(* Schneider Machine Expert - Basic project Tank_1m_Ultrasonic_TM221CE16T, file version 3.0.0.0 *)
(* ProjectInformations: Name=Tank_1m_Ultrasonic_TM221CE16T *)

HARDWARE
  Cpu 0: TM221CE16T
  ModuleExtensionObject 0: TM3AI4/G
  EthernetConfiguration: NetworkName=M221, IpAllocationMode=FixedAddress, IpAddress=0.0.0.0, SubnetMask=0.0.0.0
  SerialLineConfiguration: Baud=Baud19200, Parity=ParityEven, DataBits=DataBits8, StopBits=StopBits1, PhysicalMedium=PhysicalMediumRs485, TransmissionMode=TransmissionModeModbusRtu, SlaveId=1, Addressing=SlaveAddressing
  MastTask: UsePeriodScanMode=false, PeriodScan=100
  FastTask: Period=255
  CpuBehavior: StartingMode=StartAsPreviousState, AutoSaveRamOnEeprom=true, WatchdogPeriod=250

SYMBOLS  (address, symbol, comment, settings)
  %M0       INLET_ENABLE
  %M1       OUTLET_ENABLE
  %M2       LEVEL_HIGH
  %M3       LEVEL_LOW
  %S12      SB_RUNMODE  "The controller is running"
  %MW0      TANK_RAW  "Raw analog value from ultrasonic sensor (0-10000)"
  %MW1      TANK_LEVEL_MM  "Calculated tank level in millimeters (0-1000)"
  %MW2      TANK_LITERS  "Tank volume in liters for HMI display (0-1000L)"
  %Q0.0     INLET_VALVE
  %Q0.1     OUTLET_VALVE
  %IW1.0    ULTRASONIC_LEVEL  [Type=Type_0_10V, Scope=Scope_Normal, Minimum=0, Maximum=10000]

POU Tank Level Control
  (* SectionNumber=0 *)

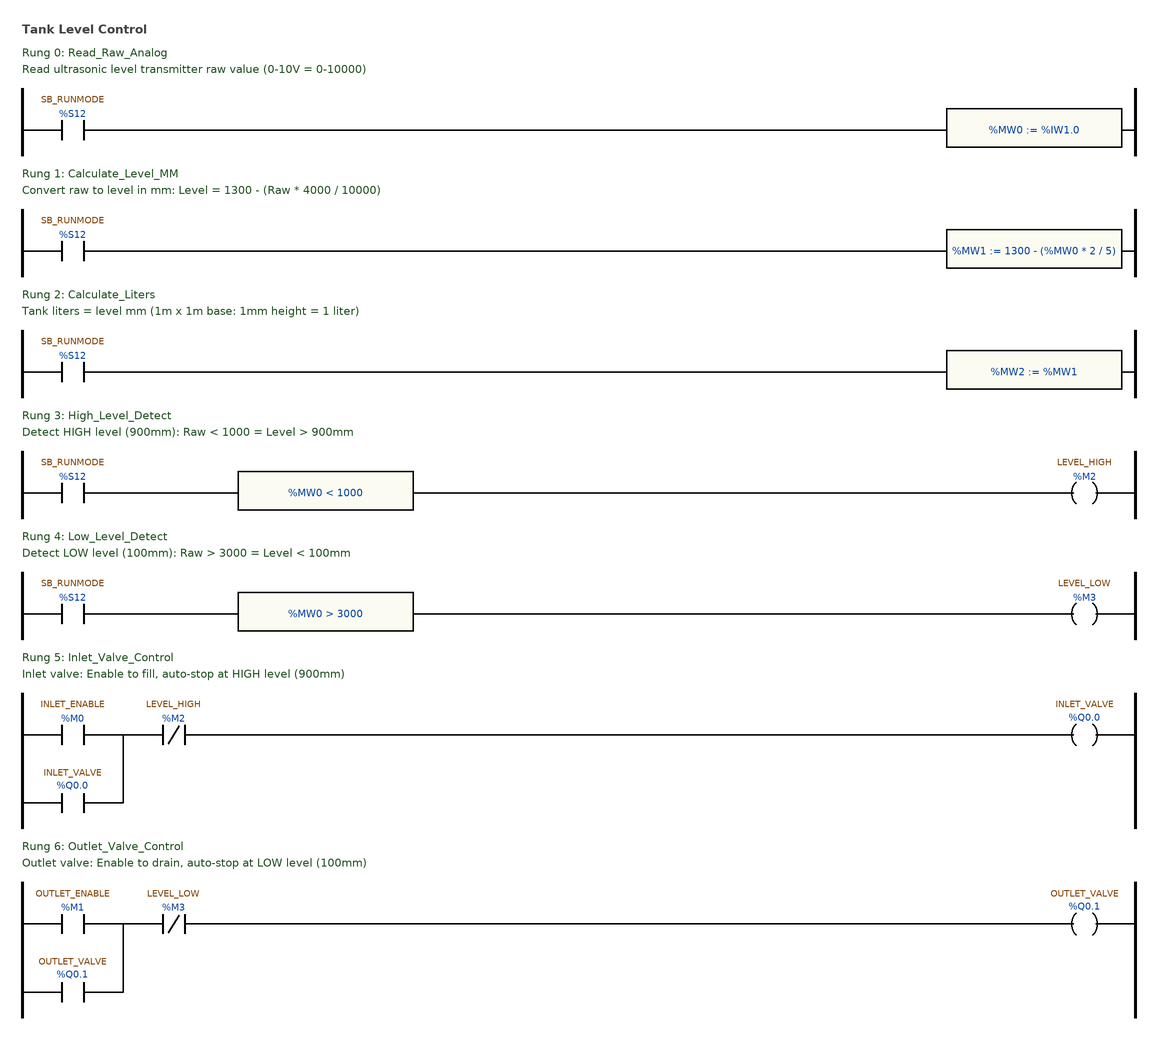

// Rung 0: Read_Raw_Analog
// Read ultrasonic level transmitter raw value (0-10V = 0-10000)
  LD %S12                 (* SB_RUNMODE *)
  [ %MW0 := %IW1.0 ]      (* TANK_RAW, ULTRASONIC_LEVEL *)
  // as ST:
  //   IF SB_RUNMODE THEN TANK_RAW := ULTRASONIC_LEVEL; END_IF;

// Rung 1: Calculate_Level_MM
// Convert raw to level in mm: Level = 1300 - (Raw * 4000 / 10000)
  LD %S12                 (* SB_RUNMODE *)
  [ %MW1 := 1300 - (%MW0 * 2 / 5) ](* TANK_LEVEL_MM, TANK_RAW *)
  // as ST:
  //   IF SB_RUNMODE THEN TANK_LEVEL_MM := 1300 - (TANK_RAW * 2 / 5); END_IF;

// Rung 2: Calculate_Liters
// Tank liters = level mm (1m x 1m base: 1mm height = 1 liter)
  LD %S12                 (* SB_RUNMODE *)
  [ %MW2 := %MW1 ]        (* TANK_LITERS, TANK_LEVEL_MM *)
  // as ST:
  //   IF SB_RUNMODE THEN TANK_LITERS := TANK_LEVEL_MM; END_IF;

// Rung 3: High_Level_Detect
// Detect HIGH level (900mm): Raw < 1000 = Level > 900mm
  LD %S12                 (* SB_RUNMODE *)
  AND [ %MW0 < 1000 ]     (* TANK_RAW *)
  ST %M2                  (* LEVEL_HIGH *)
  // as ST:
  //   LEVEL_HIGH := SB_RUNMODE AND TANK_RAW < 1000;

// Rung 4: Low_Level_Detect
// Detect LOW level (100mm): Raw > 3000 = Level < 100mm
  LD %S12                 (* SB_RUNMODE *)
  AND [ %MW0 > 3000 ]     (* TANK_RAW *)
  ST %M3                  (* LEVEL_LOW *)
  // as ST:
  //   LEVEL_LOW := SB_RUNMODE AND TANK_RAW > 3000;

// Rung 5: Inlet_Valve_Control
// Inlet valve: Enable to fill, auto-stop at HIGH level (900mm)
  LD %M0                  (* INLET_ENABLE *)
  OR %Q0.0                (* INLET_VALVE *)
  ANDN %M2                (* LEVEL_HIGH *)
  ST %Q0.0                (* INLET_VALVE *)
  // as ST:
  //   INLET_VALVE := (INLET_ENABLE OR INLET_VALVE) AND NOT LEVEL_HIGH;

// Rung 6: Outlet_Valve_Control
// Outlet valve: Enable to drain, auto-stop at LOW level (100mm)
  LD %M1                  (* OUTLET_ENABLE *)
  OR %Q0.1                (* OUTLET_VALVE *)
  ANDN %M3                (* LEVEL_LOW *)
  ST %Q0.1                (* OUTLET_VALVE *)
  // as ST:
  //   OUTLET_VALVE := (OUTLET_ENABLE OR OUTLET_VALVE) AND NOT LEVEL_LOW;
